{attribute 'qualified_only'}
VAR_GLOBAL
	
	 
	Uitgang1 AT %QX26.0 : BOOL := FALSE;
	Uitgang2 AT %QX26.1 : BOOL := FALSE;
	Uitgang3 AT %QX26.2 : BOOL := FALSE;
	Uitgang4 AT %QX26.3 : BOOL := FALSE;
	
END_VAR

(* stored: Version 1.1.0.1, ProductVersion 3.1.4024.12
   GVL DIDO: Id {2e427f3a-144f-4aff-8c4b-5ae56a94745e} *)
